TYPE MotionFn :
STRUCT
	Gearing						: typ_MotionGearing;
	Homing						: typ_MotionHoming;
	ManualMotion				: typ_MotionManualMotion;
	Phasing						: typ_MotionPhasing;
	PointToPoint				: typ_MotionPointToPoint;
END_STRUCT
END_TYPE

(* stored: Version 1.1.0.1, ProductVersion 3.1.4022.17
   DUT MotionFn: Id {a0ea39f5-338e-4681-81d0-3170bbdd26ed} *)
